{attribute 'GeneratedUsingTerminal: EL6201-0000-0017'}
{attribute addProperty BoxType "EL6201-0000-0017"}
{attribute addProperty Id "Slave_22A_DO0BOOL1Slave_22A_DO1BOOL1Slave_22A_DO2BOOL1Slave_22A_DO3BOOL1Slave_22B_DO0BOOL1Slave_22B_DO1BOOL1Slave_22B_DO2BOOL1Slave_22B_DO3BOOL1"}
{attribute addProperty CRC "976042318"}
{attribute addProperty Size "8"}
TYPE Slave_22_Outputs_3A2D394E :
STRUCT
	{attribute addProperty Name "Slave_22A_DO0"}
	Slave_22A_DO0 : BOOL;
	{attribute addProperty Name "Slave_22A_DO1"}
	Slave_22A_DO1 : BOOL;
	{attribute addProperty Name "Slave_22A_DO2"}
	Slave_22A_DO2 : BOOL;
	{attribute addProperty Name "Slave_22A_DO3"}
	Slave_22A_DO3 : BOOL;
	{attribute addProperty Name "Slave_22B_DO0"}
	Slave_22B_DO0 : BOOL;
	{attribute addProperty Name "Slave_22B_DO1"}
	Slave_22B_DO1 : BOOL;
	{attribute addProperty Name "Slave_22B_DO2"}
	Slave_22B_DO2 : BOOL;
	{attribute addProperty Name "Slave_22B_DO3"}
	Slave_22B_DO3 : BOOL;
END_STRUCT
END_TYPE

(* stored: Version 1.2.0.0, ProductVersion 3.1.4024.11
   DUT Slave_22_Outputs_3A2D394E: Id {db33352a-359e-4780-ad33-49f62a85865a} *)
